// TIA Portal V18 export
DATA_BLOCK "laser_centering_device_DB"   // DB4
VERSION : 0.1
// stored: AutoNumber true, DBAccessibleFromOPCUA true, InstanceOfName laser_centering_device, InstanceOfType FB
"laser_centering_device"
   // VAR_INPUT
   //    xBtn : Bool;
   //    pt_sec : Real;
   // END_VAR
   // VAR_OUTPUT
   //    yEnergize : Bool;
   // END_VAR
   // VAR RETAIN
   //    pt : Time;
   // END_VAR
   // VAR
   //    mem : Bool;
   //    clkBtn : Bool;
   //    IEC_Timer_0_Instance { S7_SetPoint := 'True'} : TON_TIME;
   //    xBtnWAS : Bool;
   //    should_energize_was : Bool;
   // END_VAR
BEGIN
END_DATA_BLOCK
